// TIA Portal V19 export
TYPE "ZSL_typeJobConditionsInterface"
// stored: Access Published, Namespace Unit3.EM1
   STRUCT
      jobStartingEnabled : Bool;
      jobHomingEnabled : Bool;
      jobMovePosEnabled : Bool;
      jobResetingEnabled : Bool;
   END_STRUCT;
END_TYPE
